(*
	Default binary sensor device.
*)
FUNCTION_BLOCK FB_SensorBinary EXTENDS FB_LinkDevice 
VAR_OUTPUT
	bValue		: BOOL; 
END_VAR

SUPER^();
bValue := Status.0;

END_FUNCTION_BLOCK

(* stored: Version 1.1.0.1, ProductVersion 3.1.4024.12
   POU FB_SensorBinary: Id {a825ddc3-4f91-07fd-3487-992ee91de2b5}, SpecialFunc None *)
